// TIA Portal V16 export
// export: Created 2020-10-15T11:58:20.887341Z, ExportSetting WithDefaults, DisplayName Totally Integrated Automation Portal, DisplayVersion V16, DisplayName TIA Portal Version Control Interface, DisplayVersion V16, DisplayName TIA Portal Openness, DisplayVersion V16, DisplayName STEP 7 Professional, DisplayVersion V16, DisplayName STEP 7 Safety, DisplayVersion V16, DisplayName WinCC Advanced, DisplayVersion V16
VAR_GLOBAL   // PLC tag table "AI_ENERGY_METER"
   "001EK_111_KF028_PI" AT %I100.0 : "iUDT_PI_LUETZE_LOCC_BOX";   // Locc Box Inputs
   "001EK_111_KF028_PO" AT %Q100.0 : "iUDT_PO_LUETZE_LOCC_BOX";   // Locc Box Outputs / Ausgangsschnittstelle Locc-Box
   "000EEA011-KF30.2-KF30.12_PI" AT %I702.0 : "iUDT_PI_EATON_PKE-SWD-CP";   // Periphery interface inputs EATON_PKE switch / Peripherieschnittstelle Eingänge Eaton PKE switch
   "000EE_001-KF24_1_PI" AT %I1000.0 : "iUDT_PI_AI_ENERGY_METER";   // Periphery interface inputs AI energy meter / Peripherieschnittstelle Eingänge AI Energy Meter
   "000EEA011-KF30.2-KF30.12_PO" AT %Q702.0 : "iUDT_PO_EATON_PKE-SWD-CP";   // Periphery output Eaton PKE protection switch / Peripherieausgang Eaton PKE Schutzschalter
   "000EE_001-KF24_1_PO" AT %Q1000.0 : "iUDT_PO_AI_ENERGY_METER";   // Periphery interface outputs AI energy meter / Peripherieschnittstelle Ausgänge AI Energy Meter
END_VAR
